{attribute 'GeneratedUsingTerminal: EP9224-0037-0017'}
{attribute addProperty BoxType "EP9224-0037-0017"}
{attribute addProperty Id "Warning_TemperatureBOOL1Error_TemperatureBOOL1Warning_UsBOOL1Error_UsBOOL1Warning_UpBOOL1Error_UpBOOL1Global_Error_BitBOOL1Warning_Sum_CurrentBOOL1Error_Sum_CurrentBOOL1TxPDO_StateBOOL1TxPDO_ToggleBOOL1"}
{attribute addProperty CRC "54290665"}
{attribute addProperty Size "11"}
TYPE Device_Status_033C68E9 :
STRUCT
	{attribute addProperty Name "Warning_Temperature"}
	Warning_Temperature : BOOL;
	{attribute addProperty Name "Error_Temperature"}
	Error_Temperature : BOOL;
	{attribute addProperty Name "Warning_Us"}
	Warning_Us : BOOL;
	{attribute addProperty Name "Error_Us"}
	Error_Us : BOOL;
	{attribute addProperty Name "Warning_Up"}
	Warning_Up : BOOL;
	{attribute addProperty Name "Error_Up"}
	Error_Up : BOOL;
	{attribute addProperty Name "Global_Error_Bit"}
	Global_Error_Bit : BOOL;
	{attribute addProperty Name "Warning_Sum_Current"}
	Warning_Sum_Current : BOOL;
	{attribute addProperty Name "Error_Sum_Current"}
	Error_Sum_Current : BOOL;
	{attribute addProperty Name "TxPDO_State"}
	TxPDO_State : BOOL;
	{attribute addProperty Name "TxPDO_Toggle"}
	TxPDO_Toggle : BOOL;
END_STRUCT
END_TYPE

(* stored: Version 1.2.0.0, ProductVersion 3.1.4024.11
   DUT Device_Status_033C68E9: Id {57c2e11c-8ec7-4ef9-bfe4-06c3dbf4b944} *)
